PROGRAM MAIN

{region generated code}
VAR_INPUT
	bInitRun : BOOL := TRUE;
	fbSystem : FB_System;
	FG_01 : FG_01;
	FG_02 : FG_02;
	FG_03 : FG_03;
	FG_04 : FG_04;
	FG_05 : FG_05;
	FG_System : FG_System;
	FG_Transport : FG_Transport;
END_VAR
{endregion}

{region generated code}
	InitRun();
	fbSystem();
	PRG_EtherCAT_1_SIM();
	FG_01();
	FG_02();
	FG_03();
	FG_04();
	FG_05();
	FG_System();
	FG_Transport();
{endregion}

METHOD InitRun
{region generated code}
	IF NOT bInitRun THEN RETURN; END_IF
	bInitRun := FALSE;
{endregion}
END_METHOD

END_PROGRAM

(* stored: Version 1.1.0.1, ProductVersion 3.1.4026.19
   POU MAIN: Id {dad680ec-4ae4-426d-a3b8-23551819b713}, SpecialFunc None
   Method InitRun: Id {fdf32ae9-4714-4c4b-963e-a9705ad3f334} *)
